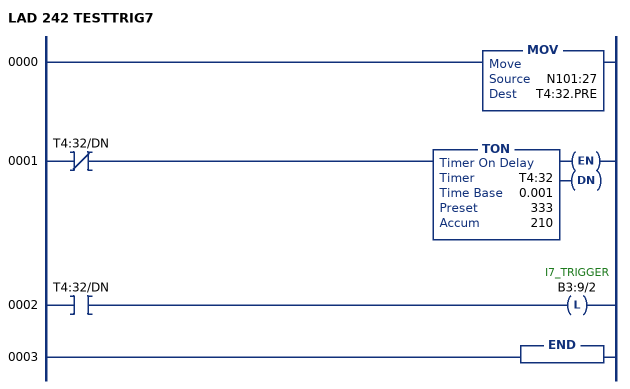
% Rung: 0 %
SOR MOV N101:27 T4:32.PRE EOR
%   N101:27  I7_TRIGTIME %
% Rung: 1 %
SOR XIO T4:32/DN TON T4:32 0.001 333 210 EOR
% Rung: 2 %
SOR XIC T4:32/DN OTL B3:9/2 EOR
%   B3:9/2  I7_TRIGGER %
% Rung: 3 %
SOR END EOR

LADDER 243 "TESTTRIG8"
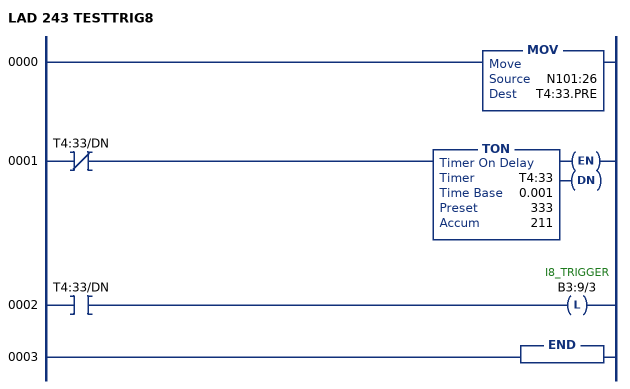
% Rung: 0 %
SOR MOV N101:26 T4:33.PRE EOR
%   N101:26  I8_TRIGTIME %
% Rung: 1 %
SOR XIO T4:33/DN TON T4:33 0.001 333 211 EOR
% Rung: 2 %
SOR XIC T4:33/DN OTL B3:9/3 EOR
%   B3:9/3  I8_TRIGGER %
% Rung: 3 %
SOR END EOR

LADDER 244 "PACKAGER"    % normal %
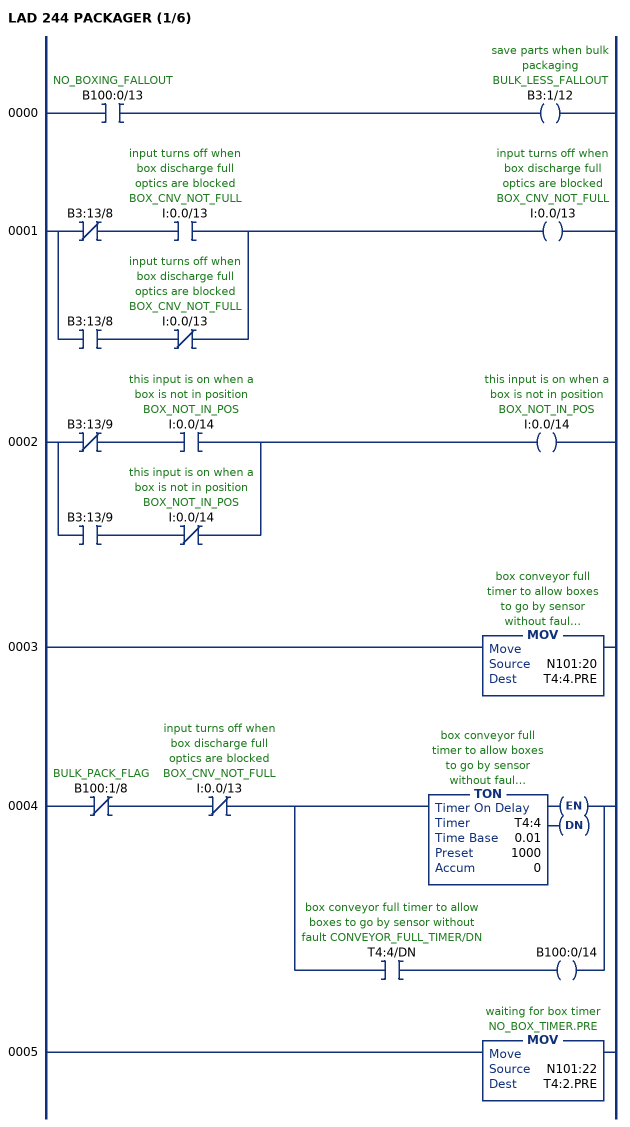
% Rung: 0 %
SOR XIC B100:0/13 OTE B3:1/12 EOR
%   B100:0/13  NO_BOXING_FALLOUT %
%   B3:1/12  BULK_LESS_FALLOUT  "save parts when bulk packaging" %
% Rung: 1 %
SOR BST XIO B3:13/8 XIC I:0.0/13 NXB XIC B3:13/8 XIO I:0.0/13 BND OTE I:0.0/13 EOR
%   I:0.0/13  BOX_CNV_NOT_FULL  "input turns off when box discharge full optics are blocked" %
% Rung: 2 %
SOR BST XIO B3:13/9 XIC I:0.0/14 NXB XIC B3:13/9 XIO I:0.0/14 BND OTE I:0.0/14 EOR
%   I:0.0/14  BOX_NOT_IN_POS  "this input is on when a box is not in position" %
% Rung: 3 %
SOR MOV N101:20 T4:4.PRE EOR
%   N101:20  CONV_FULL_TIME_LIMIT  "time to allow box to pass box conveyor full sensor without fault" %
%   T4:4  CONVEYOR_FULL_TIMER  "box conveyor full timer to allow boxes to go by sensor without fault" %
% Rung: 4 %
SOR XIO B100:1/8 XIO I:0.0/13 BST TON T4:4 0.01 1000 0 NXB XIC T4:4/DN OTE B100:0/14 BND EOR
%   B100:1/8  BULK_PACK_FLAG %
%   I:0.0/13  BOX_CNV_NOT_FULL  "input turns off when box discharge full optics are blocked" %
%   T4:4  CONVEYOR_FULL_TIMER  "box conveyor full timer to allow boxes to go by sensor without fault" %
% Rung: 5 %
SOR MOV N101:22 T4:2.PRE EOR
%   N101:22  BOX_WAIT_TIME_LIMIT  "the time until waiting for box message in hmi (fault)" %
%   T4:2  NO_BOX_TIMER  "waiting for box timer" %

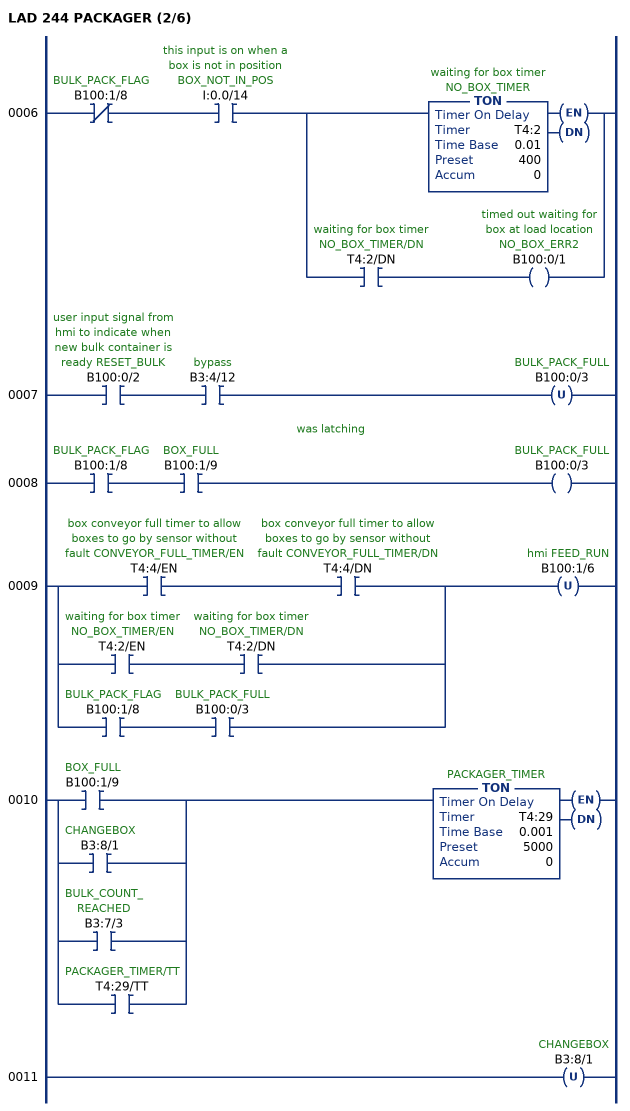
% Rung: 6 %
SOR XIO B100:1/8 XIC I:0.0/14 BST TON T4:2 0.01 400 0 NXB XIC T4:2/DN OTE B100:0/1 BND EOR
%   B100:1/8  BULK_PACK_FLAG %
%   I:0.0/14  BOX_NOT_IN_POS  "this input is on when a box is not in position" %
%   T4:2  NO_BOX_TIMER  "waiting for box timer" %
%   B100:0/1  NO_BOX_ERR2  "timed out waiting for box at load location" %
% Rung: 7 %
SOR XIC B100:0/2 XIC B3:4/12 OTU B100:0/3 EOR
%   B100:0/2  RESET_BULK  "user input signal from hmi to indicate when new bulk container is ready" %
%   B3:4/12  "bypass" %
%   B100:0/3  BULK_PACK_FULL %
% Rung: 8 %
% was latching %
SOR XIC B100:1/8 XIC B100:1/9 OTE B100:0/3 EOR
%   B100:1/8  BULK_PACK_FLAG %
%   B100:1/9  BOX_FULL %
%   B100:0/3  BULK_PACK_FULL %
% Rung: 9 %
SOR BST XIC T4:4/EN XIC T4:4/DN NXB XIC T4:2/EN XIC T4:2/DN NXB XIC B100:1/8 XIC B100:0/3 BND OTU B100:1/6 EOR
%   T4:4  CONVEYOR_FULL_TIMER  "box conveyor full timer to allow boxes to go by sensor without fault" %
%   T4:2  NO_BOX_TIMER  "waiting for box timer" %
%   B100:1/8  BULK_PACK_FLAG %
%   B100:0/3  BULK_PACK_FULL %
%   B100:1/6  FEED_RUN  "hmi" %
% Rung: 10 %
SOR BST XIC B100:1/9 NXB XIC B3:8/1 NXB XIC B3:7/3 NXB XIC T4:29/TT BND TON T4:29 0.001 5000 0 EOR
%   B100:1/9  BOX_FULL %
%   B3:8/1  CHANGEBOX %
%   B3:7/3  BULK_COUNT_REACHED %
%   T4:29  PACKAGER_TIMER %
% Rung: 11 %
SOR OTU B3:8/1 EOR
%   B3:8/1  CHANGEBOX %

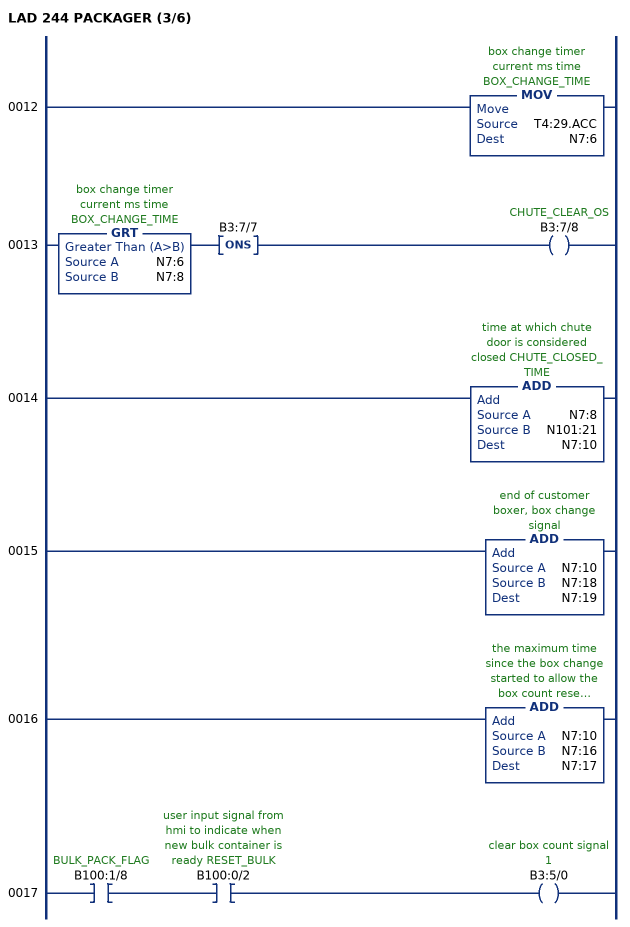
% Rung: 12 %
SOR MOV T4:29.ACC N7:6 EOR
%   T4:29  PACKAGER_TIMER %
%   N7:6  BOX_CHANGE_TIME  "box change timer current ms time" %
% Rung: 13 %
SOR GRT N7:6 N7:8 ONS B3:7/7 OTE B3:7/8 EOR
%   N7:6  BOX_CHANGE_TIME  "box change timer current ms time" %
%   N7:8  CHUTE_CLEAR_TIME %
%   B3:7/8  CHUTE_CLEAR_OS %
% Rung: 14 %
SOR ADD N7:8 N101:21 N7:10 EOR
%   N7:8  CHUTE_CLEAR_TIME %
%   N101:21  CHUTE_CLOSE_TIME  "ms time required to close chute" %
%   N7:10  CHUTE_CLOSED_TIME  "time at which chute door is considered closed" %
% Rung: 15 %
SOR ADD N7:10 N7:18 N7:19 EOR
%   N7:10  CHUTE_CLOSED_TIME  "time at which chute door is considered closed" %
%   N7:18  CHANGE_BOX_SIG_TIME  "customer boxer change box signal time" %
%   N7:19  "end of customer boxer, box change signal" %
% Rung: 16 %
SOR ADD N7:10 N7:16 N7:17 EOR
%   N7:10  CHUTE_CLOSED_TIME  "time at which chute door is considered closed" %
%   N7:16  RESET_COUNT_SIG_TIME  "maximum length of time to hold box count reset signal on" %
%   N7:17  "the maximum time since the box change started to allow the box count reset signal" %
% Rung: 17 %
SOR XIC B100:1/8 XIC B100:0/2 OTE B3:5/0 EOR
%   B100:1/8  BULK_PACK_FLAG %
%   B100:0/2  RESET_BULK  "user input signal from hmi to indicate when new bulk container is ready" %
%   B3:5/0  "clear box count signal 1" %

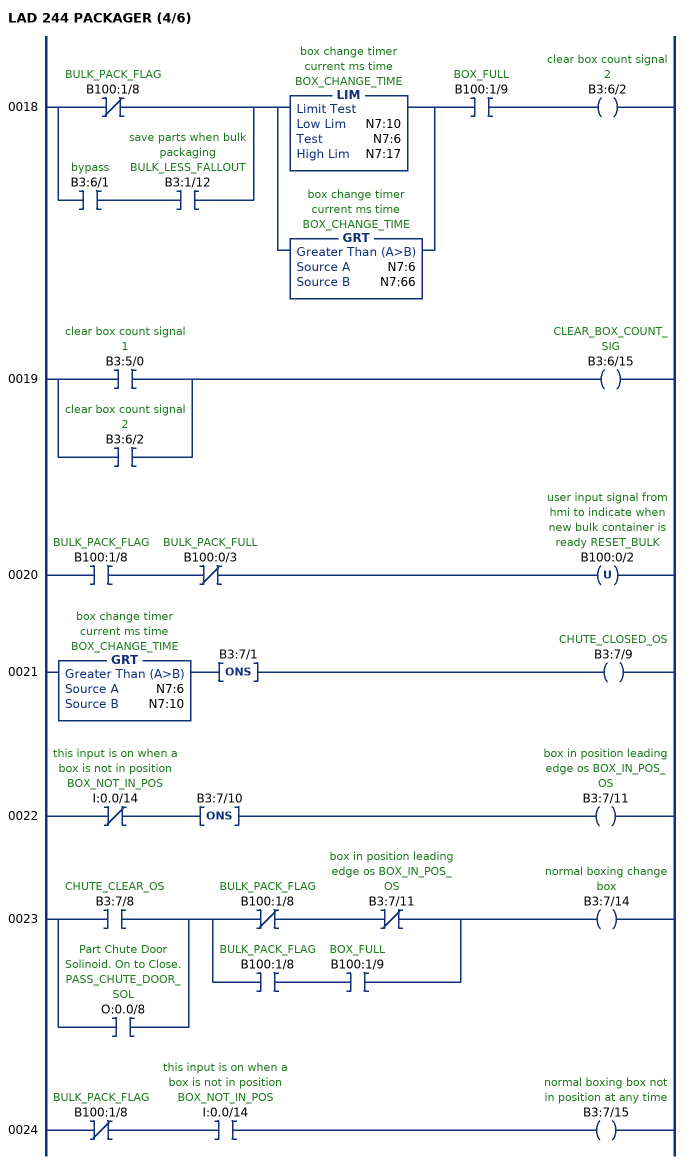
% Rung: 18 %
SOR BST XIO B100:1/8 NXB XIC B3:6/1 XIC B3:1/12 BND BST LIM N7:10 N7:6 N7:17 NXB GRT N7:6 N7:66 BND XIC B100:1/9 OTE B3:6/2 EOR
%   B100:1/8  BULK_PACK_FLAG %
%   B3:6/1  "bypass" %
%   B3:1/12  BULK_LESS_FALLOUT  "save parts when bulk packaging" %
%   N7:10  CHUTE_CLOSED_TIME  "time at which chute door is considered closed" %
%   N7:6  BOX_CHANGE_TIME  "box change timer current ms time" %
%   N7:17  "the maximum time since the box change started to allow the box count reset signal" %
%   B100:1/9  BOX_FULL %
%   B3:6/2  "clear box count signal 2" %
% Rung: 19 %
SOR BST XIC B3:5/0 NXB XIC B3:6/2 BND OTE B3:6/15 EOR
%   B3:5/0  "clear box count signal 1" %
%   B3:6/2  "clear box count signal 2" %
%   B3:6/15  CLEAR_BOX_COUNT_SIG %
% Rung: 20 %
SOR XIC B100:1/8 XIO B100:0/3 OTU B100:0/2 EOR
%   B100:1/8  BULK_PACK_FLAG %
%   B100:0/3  BULK_PACK_FULL %
%   B100:0/2  RESET_BULK  "user input signal from hmi to indicate when new bulk container is ready" %
% Rung: 21 %
SOR GRT N7:6 N7:10 ONS B3:7/1 OTE B3:7/9 EOR
%   N7:6  BOX_CHANGE_TIME  "box change timer current ms time" %
%   N7:10  CHUTE_CLOSED_TIME  "time at which chute door is considered closed" %
%   B3:7/9  CHUTE_CLOSED_OS %
% Rung: 22 %
SOR XIO I:0.0/14 ONS B3:7/10 OTE B3:7/11 EOR
%   I:0.0/14  BOX_NOT_IN_POS  "this input is on when a box is not in position" %
%   B3:7/11  BOX_IN_POS_OS  "box in position leading edge os" %
% Rung: 23 %
SOR BST XIC B3:7/8 NXB XIC O:0.0/8 BND BST XIO B100:1/8 XIO B3:7/11 NXB XIC B100:1/8 XIC B100:1/9 BND OTE B3:7/14 EOR
%   B3:7/8  CHUTE_CLEAR_OS %
%   O:0.0/8  PASS_CHUTE_DOOR_SOL  "Part Chute Door Solinoid. On to Close." %
%   B100:1/8  BULK_PACK_FLAG %
%   B3:7/11  BOX_IN_POS_OS  "box in position leading edge os" %
%   B100:1/9  BOX_FULL %
%   B3:7/14  "normal boxing change box" %
% Rung: 24 %
SOR XIO B100:1/8 XIC I:0.0/14 OTE B3:7/15 EOR
%   B100:1/8  BULK_PACK_FLAG %
%   I:0.0/14  BOX_NOT_IN_POS  "this input is on when a box is not in position" %
%   B3:7/15  "normal boxing box not in position at any time" %

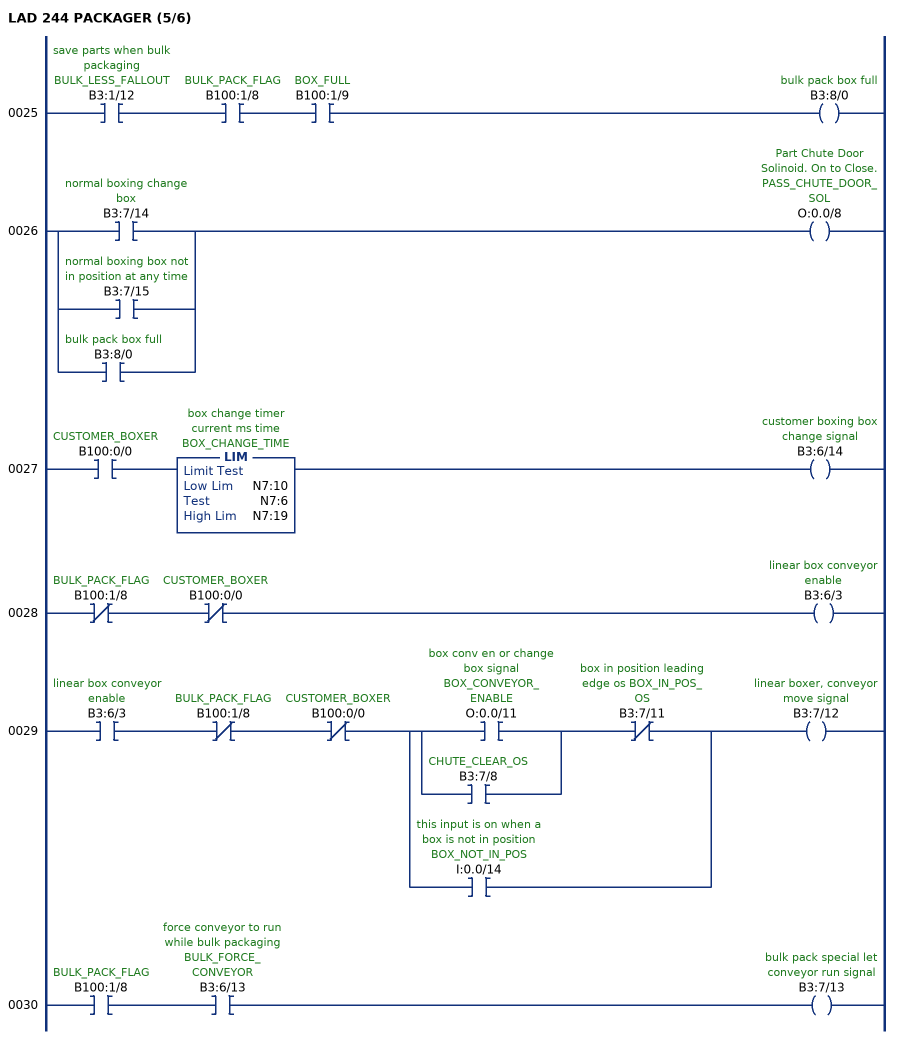
% Rung: 25 %
SOR XIC B3:1/12 XIC B100:1/8 XIC B100:1/9 OTE B3:8/0 EOR
%   B3:1/12  BULK_LESS_FALLOUT  "save parts when bulk packaging" %
%   B100:1/8  BULK_PACK_FLAG %
%   B100:1/9  BOX_FULL %
%   B3:8/0  "bulk pack box full" %
% Rung: 26 %
SOR BST XIC B3:7/14 NXB XIC B3:7/15 NXB XIC B3:8/0 BND OTE O:0.0/8 EOR
%   B3:7/14  "normal boxing change box" %
%   B3:7/15  "normal boxing box not in position at any time" %
%   B3:8/0  "bulk pack box full" %
%   O:0.0/8  PASS_CHUTE_DOOR_SOL  "Part Chute Door Solinoid. On to Close." %
% Rung: 27 %
SOR XIC B100:0/0 LIM N7:10 N7:6 N7:19 OTE B3:6/14 EOR
%   B100:0/0  CUSTOMER_BOXER %
%   N7:10  CHUTE_CLOSED_TIME  "time at which chute door is considered closed" %
%   N7:6  BOX_CHANGE_TIME  "box change timer current ms time" %
%   N7:19  "end of customer boxer, box change signal" %
%   B3:6/14  "customer boxing box change signal" %
% Rung: 28 %
SOR XIO B100:1/8 XIO B100:0/0 OTE B3:6/3 EOR
%   B100:1/8  BULK_PACK_FLAG %
%   B100:0/0  CUSTOMER_BOXER %
%   B3:6/3  "linear box conveyor enable" %
% Rung: 29 %
SOR XIC B3:6/3 XIO B100:1/8 XIO B100:0/0 BST BST XIC O:0.0/11 NXB XIC B3:7/8 BND XIO B3:7/11 NXB XIC I:0.0/14 BND OTE B3:7/12 EOR
%   B3:6/3  "linear box conveyor enable" %
%   B100:1/8  BULK_PACK_FLAG %
%   B100:0/0  CUSTOMER_BOXER %
%   O:0.0/11  BOX_CONVEYOR_ENABLE  "box conv en or change box signal" %
%   B3:7/8  CHUTE_CLEAR_OS %
%   B3:7/11  BOX_IN_POS_OS  "box in position leading edge os" %
%   I:0.0/14  BOX_NOT_IN_POS  "this input is on when a box is not in position" %
%   B3:7/12  "linear boxer, conveyor move signal" %
% Rung: 30 %
SOR XIC B100:1/8 XIC B3:6/13 OTE B3:7/13 EOR
%   B100:1/8  BULK_PACK_FLAG %
%   B3:6/13  BULK_FORCE_CONVEYOR  "force conveyor to run while bulk packaging" %
%   B3:7/13  "bulk pack special let conveyor run signal" %

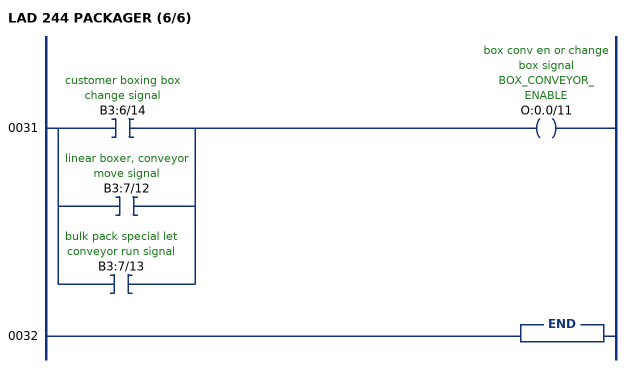
% Rung: 31 %
SOR BST XIC B3:6/14 NXB XIC B3:7/12 NXB XIC B3:7/13 BND OTE O:0.0/11 EOR
%   B3:6/14  "customer boxing box change signal" %
%   B3:7/12  "linear boxer, conveyor move signal" %
%   B3:7/13  "bulk pack special let conveyor run signal" %
%   O:0.0/11  BOX_CONVEYOR_ENABLE  "box conv en or change box signal" %
% Rung: 32 %
SOR END EOR

LADDER 245 "NO PACKAGE"
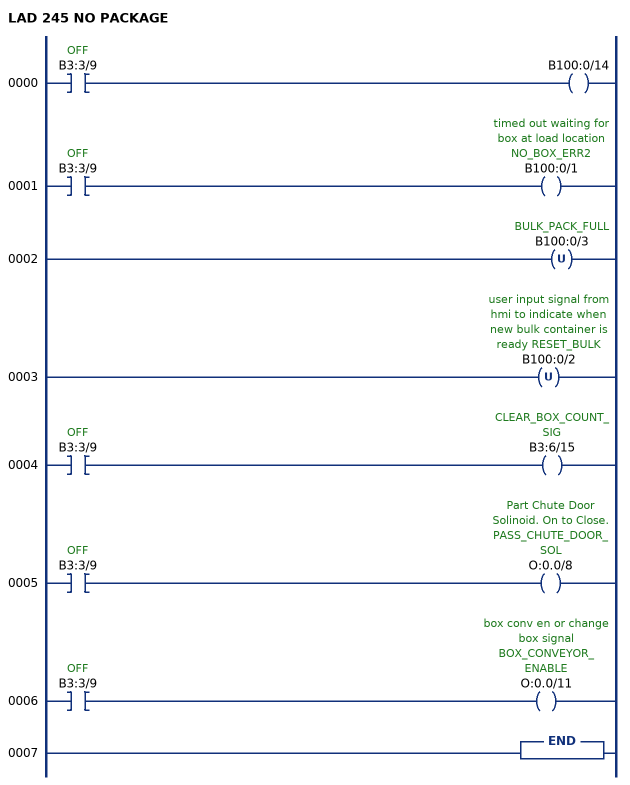
% Rung: 0 %
SOR XIC B3:3/9 OTE B100:0/14 EOR
%   B3:3/9  OFF %
% Rung: 1 %
SOR XIC B3:3/9 OTE B100:0/1 EOR
%   B3:3/9  OFF %
%   B100:0/1  NO_BOX_ERR2  "timed out waiting for box at load location" %
% Rung: 2 %
SOR OTU B100:0/3 EOR
%   B100:0/3  BULK_PACK_FULL %
% Rung: 3 %
SOR OTU B100:0/2 EOR
%   B100:0/2  RESET_BULK  "user input signal from hmi to indicate when new bulk container is ready" %
% Rung: 4 %
SOR XIC B3:3/9 OTE B3:6/15 EOR
%   B3:3/9  OFF %
%   B3:6/15  CLEAR_BOX_COUNT_SIG %
% Rung: 5 %
SOR XIC B3:3/9 OTE O:0.0/8 EOR
%   B3:3/9  OFF %
%   O:0.0/8  PASS_CHUTE_DOOR_SOL  "Part Chute Door Solinoid. On to Close." %
% Rung: 6 %
SOR XIC B3:3/9 OTE O:0.0/11 EOR
%   B3:3/9  OFF %
%   O:0.0/11  BOX_CONVEYOR_ENABLE  "box conv en or change box signal" %
% Rung: 7 %
SOR END EOR

LADDER 246 "RATE1"
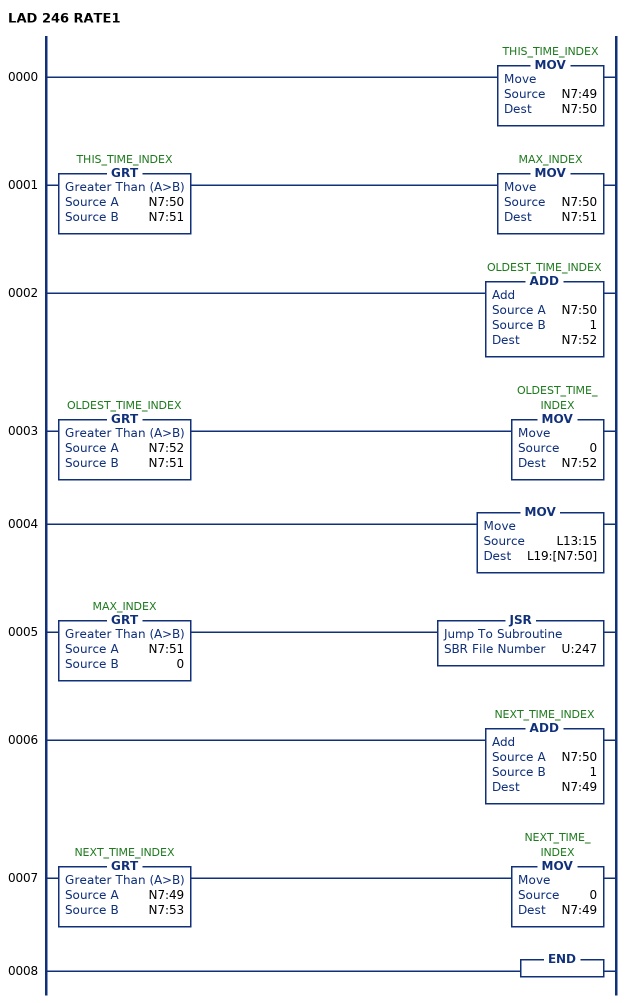
% Rung: 0 %
SOR MOV N7:49 N7:50 EOR
%   N7:49  NEXT_TIME_INDEX %
%   N7:50  THIS_TIME_INDEX %
% Rung: 1 %
SOR GRT N7:50 N7:51 MOV N7:50 N7:51 EOR
%   N7:50  THIS_TIME_INDEX %
%   N7:51  MAX_INDEX %
% Rung: 2 %
SOR ADD N7:50 1 N7:52 EOR
%   N7:50  THIS_TIME_INDEX %
%   N7:52  OLDEST_TIME_INDEX %
% Rung: 3 %
SOR GRT N7:52 N7:51 MOV 0 N7:52 EOR
%   N7:52  OLDEST_TIME_INDEX %
%   N7:51  MAX_INDEX %
% Rung: 4 %
SOR MOV L13:15 L19:[N7:50] EOR
%   L13:15  THE_TIME %
%   N7:50  THIS_TIME_INDEX %
% Rung: 5 %
SOR GRT N7:51 0 JSR U:247 EOR
%   N7:51  MAX_INDEX %
% Rung: 6 %
SOR ADD N7:50 1 N7:49 EOR
%   N7:50  THIS_TIME_INDEX %
%   N7:49  NEXT_TIME_INDEX %
% Rung: 7 %
SOR GRT N7:49 N7:53 MOV 0 N7:49 EOR
%   N7:49  NEXT_TIME_INDEX %
%   N7:53  UPPER_INDEX_LIMIT %
% Rung: 8 %
SOR END EOR

LADDER 247 "RATE2"
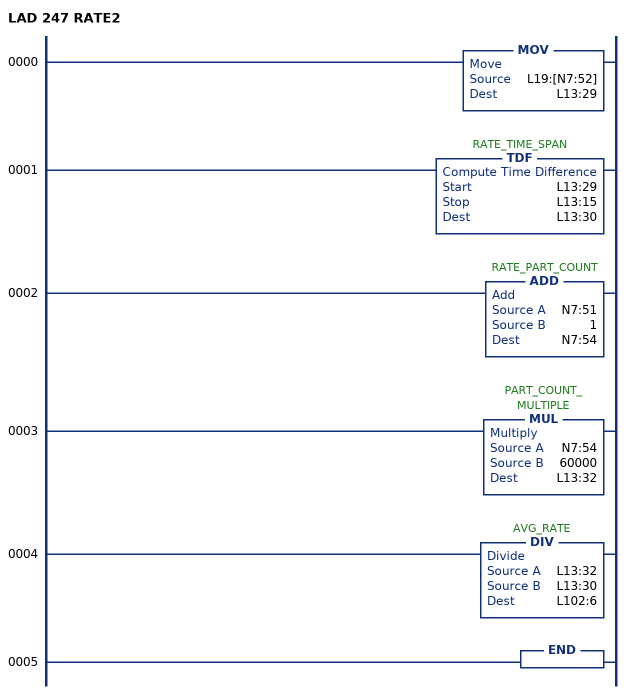
% Rung: 0 %
SOR MOV L19:[N7:52] L13:29 EOR
%   N7:52  OLDEST_TIME_INDEX %
% Rung: 1 %
SOR TDF L13:29 L13:15 L13:30 EOR
%   L13:15  THE_TIME %
%   L13:30  RATE_TIME_SPAN %
% Rung: 2 %
SOR ADD N7:51 1 N7:54 EOR
%   N7:51  MAX_INDEX %
%   N7:54  RATE_PART_COUNT %
% Rung: 3 %
SOR MUL N7:54 60000 L13:32 EOR
%   N7:54  RATE_PART_COUNT %
%   L13:32  PART_COUNT_MULTIPLE %
% Rung: 4 %
SOR DIV L13:32 L13:30 L102:6 EOR
%   L13:32  PART_COUNT_MULTIPLE %
%   L13:30  RATE_TIME_SPAN %
%   L102:6  AVG_RATE %
% Rung: 5 %
SOR END EOR

LADDER 248 "RESET RATE"
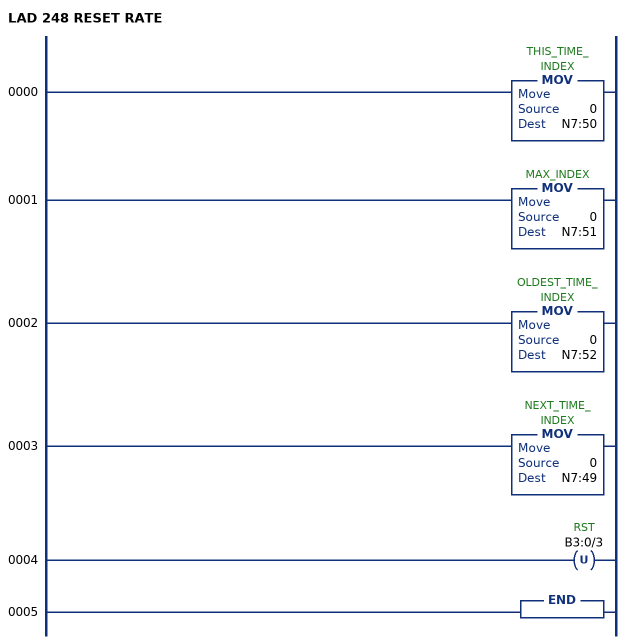
% Rung: 0 %
SOR MOV 0 N7:50 EOR
%   N7:50  THIS_TIME_INDEX %
% Rung: 1 %
SOR MOV 0 N7:51 EOR
%   N7:51  MAX_INDEX %
% Rung: 2 %
SOR MOV 0 N7:52 EOR
%   N7:52  OLDEST_TIME_INDEX %
% Rung: 3 %
SOR MOV 0 N7:49 EOR
%   N7:49  NEXT_TIME_INDEX %
% Rung: 4 %
SOR OTU B3:0/3 EOR
%   B3:0/3  RST %
% Rung: 5 %
SOR END EOR

LADDER 249 "NP STOP"    % stop on no good %
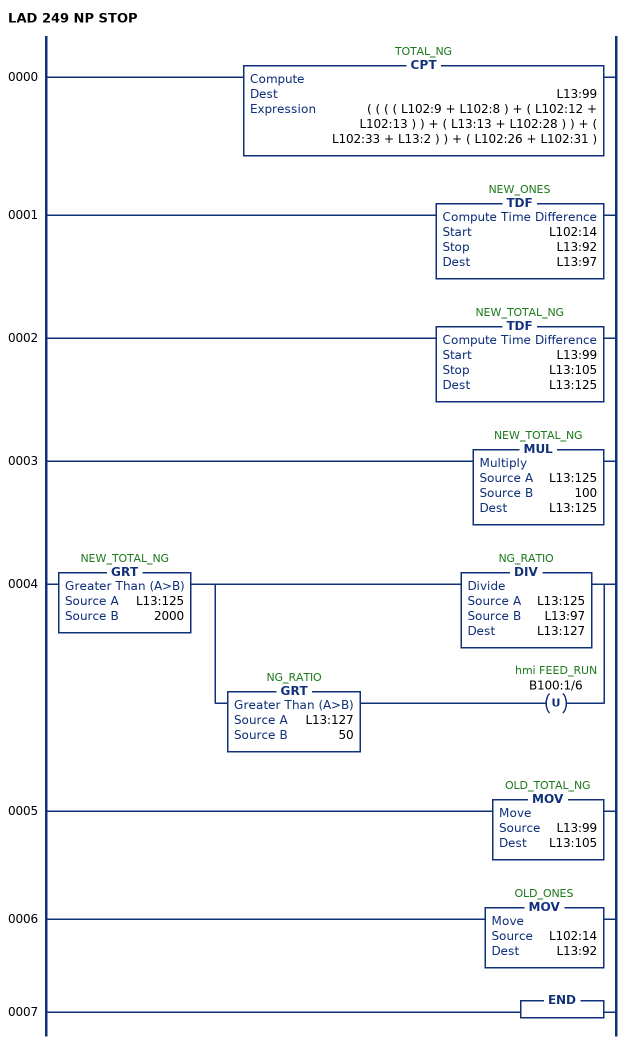
% Rung: 0 %
SOR CPT L13:99 " ( ( ( ( L102:9 + L102:8 ) + ( L102:12 + L102:13 ) ) + ( L13:13 + L102:28 ) ) + ( L102:33 + L13:2 ) ) + ( L102:26 + L102:31 ) " EOR
%   L13:99  TOTAL_NG %
%   L102:9  "too wide bottom" %
%   L102:8  "too close bottom" %
%   L102:12  "too close top count" %
%   L102:13  "too wide top count" %
%   L102:28  I1_I5_SKIPPEDCOUNT %
%   L102:33  I2_I6_SKIPPEDCOUNT %
%   L102:26  I1_I5_FAIL_COUNT %
%   L102:31  I2_I6_FAIL_COUNT %
% Rung: 1 %
SOR TDF L102:14 L13:92 L13:97 EOR
%   L102:14  ONES %
%   L13:92  OLD_ONES %
%   L13:97  NEW_ONES %
% Rung: 2 %
SOR TDF L13:99 L13:105 L13:125 EOR
%   L13:99  TOTAL_NG %
%   L13:105  OLD_TOTAL_NG %
%   L13:125  NEW_TOTAL_NG %
% Rung: 3 %
SOR MUL L13:125 100 L13:125 EOR
%   L13:125  NEW_TOTAL_NG %
% Rung: 4 %
SOR GRT L13:125 2000 BST DIV L13:125 L13:97 L13:127 NXB GRT L13:127 50 OTU B100:1/6 BND EOR
%   L13:125  NEW_TOTAL_NG %
%   L13:97  NEW_ONES %
%   L13:127  NG_RATIO %
%   B100:1/6  FEED_RUN  "hmi" %
% Rung: 5 %
SOR MOV L13:99 L13:105 EOR
%   L13:99  TOTAL_NG %
%   L13:105  OLD_TOTAL_NG %
% Rung: 6 %
SOR MOV L102:14 L13:92 EOR
%   L102:14  ONES %
%   L13:92  OLD_ONES %
% Rung: 7 %
SOR END EOR

LADDER 250 "SPEED BOT"    % high speed %
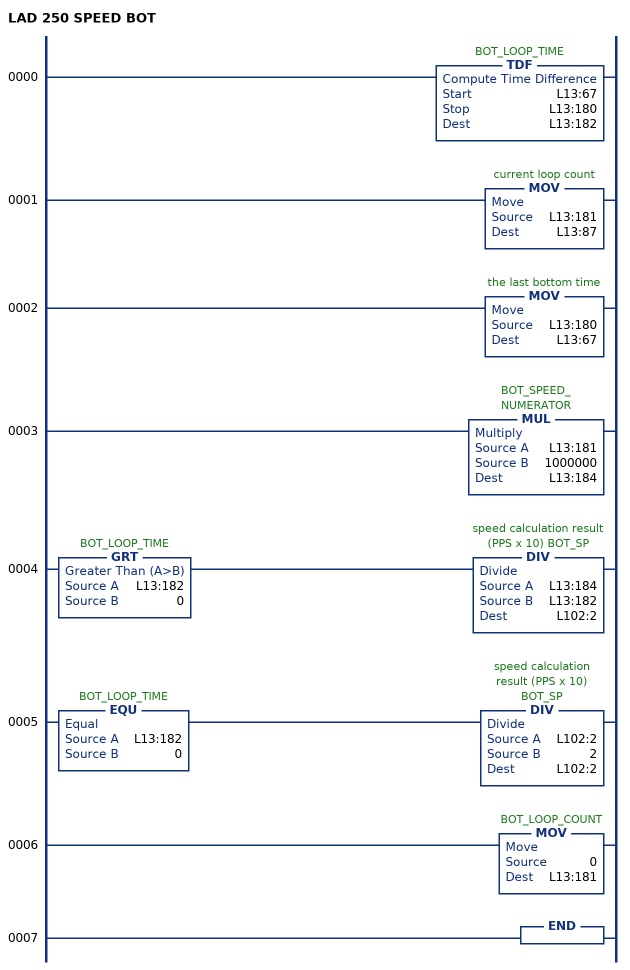
% Rung: 0 %
SOR TDF L13:67 L13:180 L13:182 EOR
%   L13:67  "the last bottom time" %
%   L13:180  BOT_THIS_TIME  "rtc bot belt movement event time" %
%   L13:182  BOT_LOOP_TIME %
% Rung: 1 %
SOR MOV L13:181 L13:87 EOR
%   L13:181  BOT_LOOP_COUNT %
%   L13:87  "current loop count" %
% Rung: 2 %
SOR MOV L13:180 L13:67 EOR
%   L13:180  BOT_THIS_TIME  "rtc bot belt movement event time" %
%   L13:67  "the last bottom time" %
% Rung: 3 %
SOR MUL L13:181 1000000 L13:184 EOR
%   L13:181  BOT_LOOP_COUNT %
%   L13:184  BOT_SPEED_NUMERATOR %
% Rung: 4 %
SOR GRT L13:182 0 DIV L13:184 L13:182 L102:2 EOR
%   L13:182  BOT_LOOP_TIME %
%   L13:184  BOT_SPEED_NUMERATOR %
%   L102:2  BOT_SP  "speed calculation result (PPS x 10)" %
% Rung: 5 %
SOR EQU L13:182 0 DIV L102:2 2 L102:2 EOR
%   L13:182  BOT_LOOP_TIME %
%   L102:2  BOT_SP  "speed calculation result (PPS x 10)" %
% Rung: 6 %
SOR MOV 0 L13:181 EOR
%   L13:181  BOT_LOOP_COUNT %
% Rung: 7 %
SOR END EOR

LADDER 251 "SPEED TOP"    % high speed %
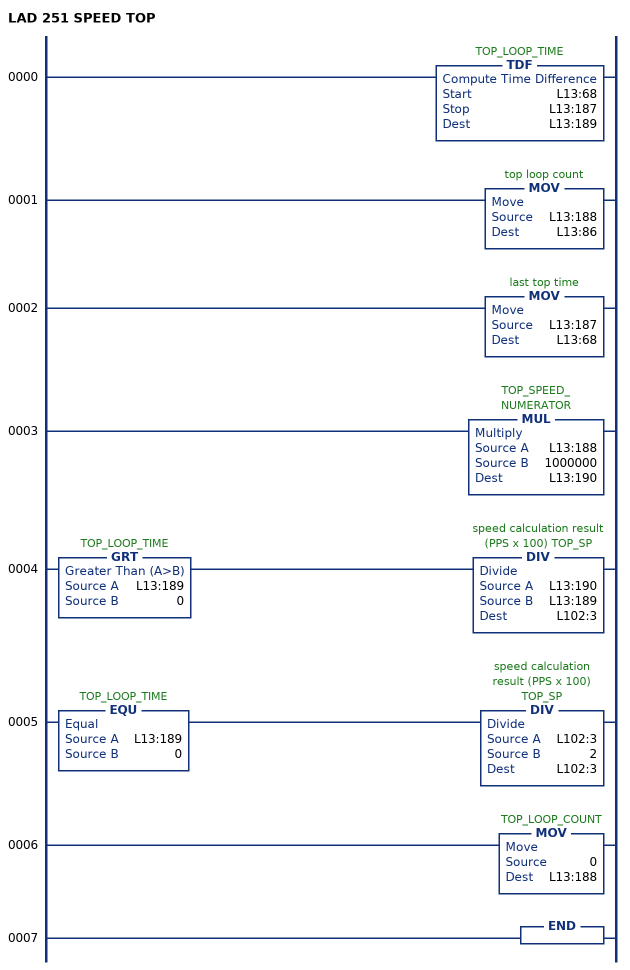
% Rung: 0 %
SOR TDF L13:68 L13:187 L13:189 EOR
%   L13:68  "last top time" %
%   L13:187  TOP_THIS_TIME  "rtc top belt movement event time" %
%   L13:189  TOP_LOOP_TIME %
% Rung: 1 %
SOR MOV L13:188 L13:86 EOR
%   L13:188  TOP_LOOP_COUNT %
%   L13:86  "top loop count" %
% Rung: 2 %
SOR MOV L13:187 L13:68 EOR
%   L13:187  TOP_THIS_TIME  "rtc top belt movement event time" %
%   L13:68  "last top time" %
% Rung: 3 %
SOR MUL L13:188 1000000 L13:190 EOR
%   L13:188  TOP_LOOP_COUNT %
%   L13:190  TOP_SPEED_NUMERATOR %
% Rung: 4 %
SOR GRT L13:189 0 DIV L13:190 L13:189 L102:3 EOR
%   L13:189  TOP_LOOP_TIME %
%   L13:190  TOP_SPEED_NUMERATOR %
%   L102:3  TOP_SP  "speed calculation result (PPS x 100)" %
% Rung: 5 %
SOR EQU L13:189 0 DIV L102:3 2 L102:3 EOR
%   L13:189  TOP_LOOP_TIME %
%   L102:3  TOP_SP  "speed calculation result (PPS x 100)" %
% Rung: 6 %
SOR MOV 0 L13:188 EOR
%   L13:188  TOP_LOOP_COUNT %
% Rung: 7 %
SOR END EOR

LADDER 252 "P BOT"    % high speed %
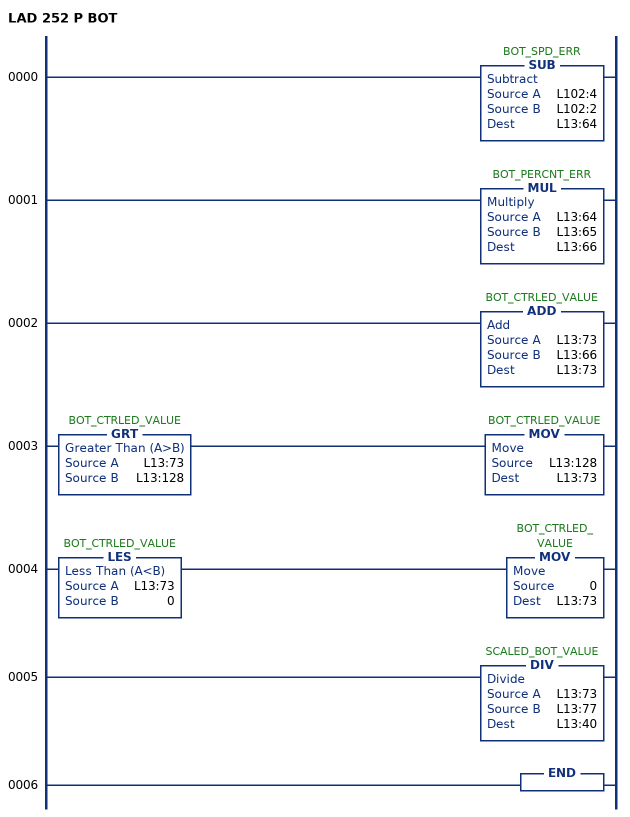
% Rung: 0 %
SOR SUB L102:4 L102:2 L13:64 EOR
%   L102:4  BOT_SPD_SETPOINT %
%   L102:2  BOT_SP  "speed calculation result (PPS x 10)" %
%   L13:64  BOT_SPD_ERR %
% Rung: 1 %
SOR MUL L13:64 L13:65 L13:66 EOR
%   L13:64  BOT_SPD_ERR %
%   L13:65  POS5SHIFT %
%   L13:66  BOT_PERCNT_ERR %
% Rung: 2 %
SOR ADD L13:73 L13:66 L13:73 EOR
%   L13:73  BOT_CTRLED_VALUE %
%   L13:66  BOT_PERCNT_ERR %
% Rung: 3 %
SOR GRT L13:73 L13:128 MOV L13:128 L13:73 EOR
%   L13:73  BOT_CTRLED_VALUE %
%   L13:128  "how much top has shifted since measurment" %
% Rung: 4 %
SOR LES L13:73 0 MOV 0 L13:73 EOR
%   L13:73  BOT_CTRLED_VALUE %
% Rung: 5 %
SOR DIV L13:73 L13:77 L13:40 EOR
%   L13:73  BOT_CTRLED_VALUE %
%   L13:40  SCALED_BOT_VALUE %
% Rung: 6 %
SOR END EOR

LADDER 253 "P TOP"    % high speed %
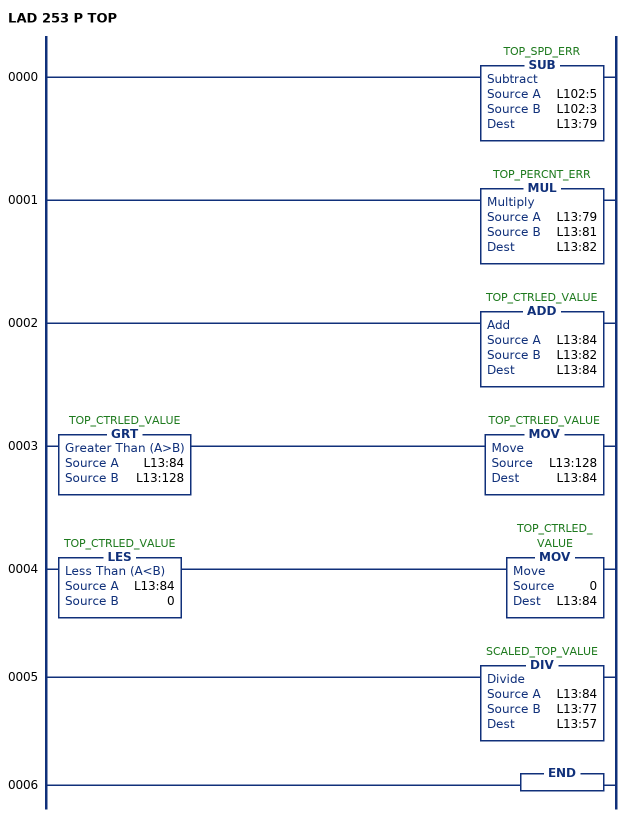
% Rung: 0 %
SOR SUB L102:5 L102:3 L13:79 EOR
%   L102:5  TOP_SPD_SETPOINT %
%   L102:3  TOP_SP  "speed calculation result (PPS x 100)" %
%   L13:79  TOP_SPD_ERR %
% Rung: 1 %
SOR MUL L13:79 L13:81 L13:82 EOR
%   L13:79  TOP_SPD_ERR %
%   L13:81  TOP_FDBK_RATIO %
%   L13:82  TOP_PERCNT_ERR %
% Rung: 2 %
SOR ADD L13:84 L13:82 L13:84 EOR
%   L13:84  TOP_CTRLED_VALUE %
%   L13:82  TOP_PERCNT_ERR %
% Rung: 3 %
SOR GRT L13:84 L13:128 MOV L13:128 L13:84 EOR
%   L13:84  TOP_CTRLED_VALUE %
%   L13:128  "how much top has shifted since measurment" %
% Rung: 4 %
SOR LES L13:84 0 MOV 0 L13:84 EOR
%   L13:84  TOP_CTRLED_VALUE %
% Rung: 5 %
SOR DIV L13:84 L13:77 L13:57 EOR
%   L13:84  TOP_CTRLED_VALUE %
%   L13:57  SCALED_TOP_VALUE %
% Rung: 6 %
SOR END EOR

LADDER 254 "TOTALCOUNT"
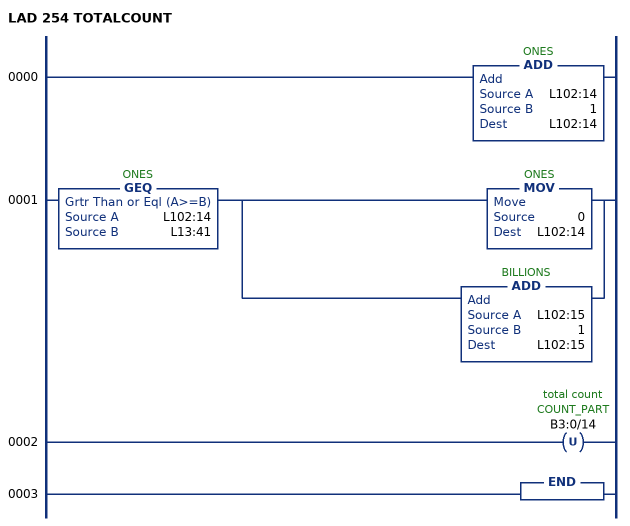
% Rung: 0 %
SOR ADD L102:14 1 L102:14 EOR
%   L102:14  ONES %
% Rung: 1 %
SOR GEQ L102:14 L13:41 BST MOV 0 L102:14 NXB ADD L102:15 1 L102:15 BND EOR
%   L102:14  ONES %
%   L13:41  "skipped count change in the last 3 seconds" %
%   L102:15  BILLIONS %
% Rung: 2 %
SOR OTU B3:0/14 EOR
%   B3:0/14  COUNT_PART  "total count" %
% Rung: 3 %
SOR END EOR

LADDER 255 "SAVED"
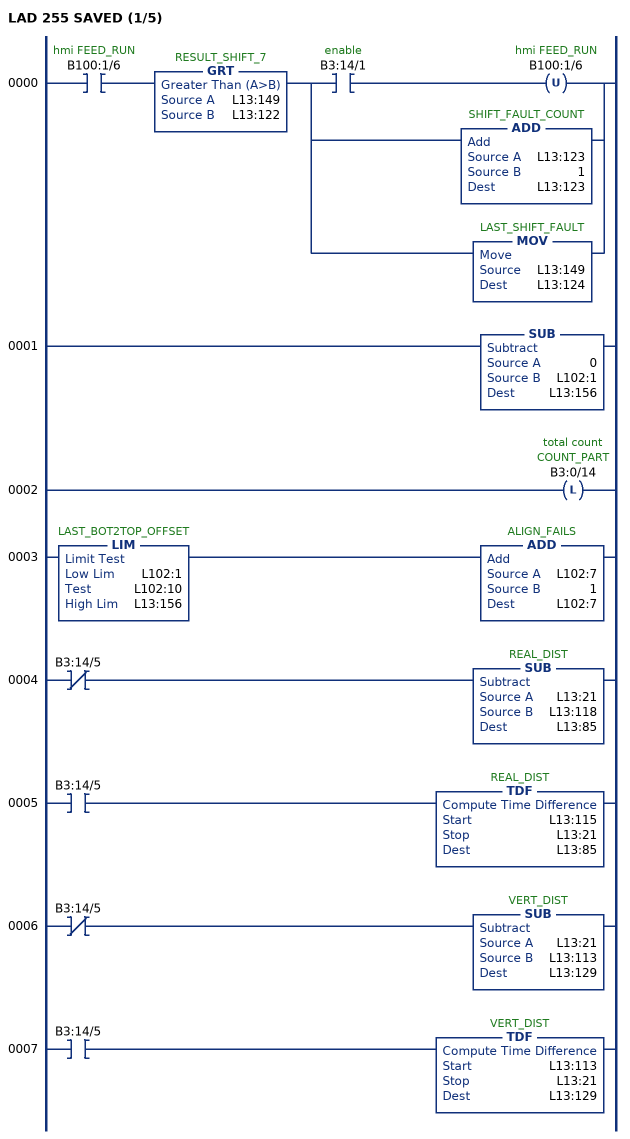
% Rung: 0 %
SOR XIC B100:1/6 GRT L13:149 L13:122 BST XIC B3:14/1 OTU B100:1/6 NXB ADD L13:123 1 L13:123 NXB MOV L13:149 L13:124 BND EOR
%   B100:1/6  FEED_RUN  "hmi" %
%   L13:149  RESULT_SHIFT_7 %
%   L13:122  TOP_SHIFT_FAULT_LIM  "remove me" %
%   B3:14/1  "enable" %
%   L13:123  SHIFT_FAULT_COUNT %
%   L13:124  LAST_SHIFT_FAULT %
% Rung: 1 %
SOR SUB 0 L102:1 L13:156 EOR
%   L102:1  MAX_OFFSET  "transition zone width" %
% Rung: 2 %
SOR OTL B3:0/14 EOR
%   B3:0/14  COUNT_PART  "total count" %
% Rung: 3 %
SOR LIM L102:1 L102:10 L13:156 ADD L102:7 1 L102:7 EOR
%   L102:1  MAX_OFFSET  "transition zone width" %
%   L102:10  LAST_BOT2TOP_OFFSET %
%   L102:7  ALIGN_FAILS %
% Rung: 4 %
SOR XIO B3:14/5 SUB L13:21 L13:118 L13:85 EOR
%   L13:21  TOP_POSITION %
%   L13:118  REAL_CL_POSITION  "real part center line in raw position" %
%   L13:85  REAL_DIST %
% Rung: 5 %
SOR XIC B3:14/5 TDF L13:115 L13:21 L13:85 EOR
%   L13:115  TRAILING_EDGE_POS  "top optic trailing edge position" %
%   L13:21  TOP_POSITION %
%   L13:85  REAL_DIST %
% Rung: 6 %
SOR XIO B3:14/5 SUB L13:21 L13:113 L13:129 EOR
%   L13:21  TOP_POSITION %
%   L13:113  VIRT_CL_POSITION  "virtual part center line transfer from the bottom in raw position" %
%   L13:129  VERT_DIST %
% Rung: 7 %
SOR XIC B3:14/5 TDF L13:113 L13:21 L13:129 EOR
%   L13:113  VIRT_CL_POSITION  "virtual part center line transfer from the bottom in raw position" %
%   L13:21  TOP_POSITION %
%   L13:129  VERT_DIST %

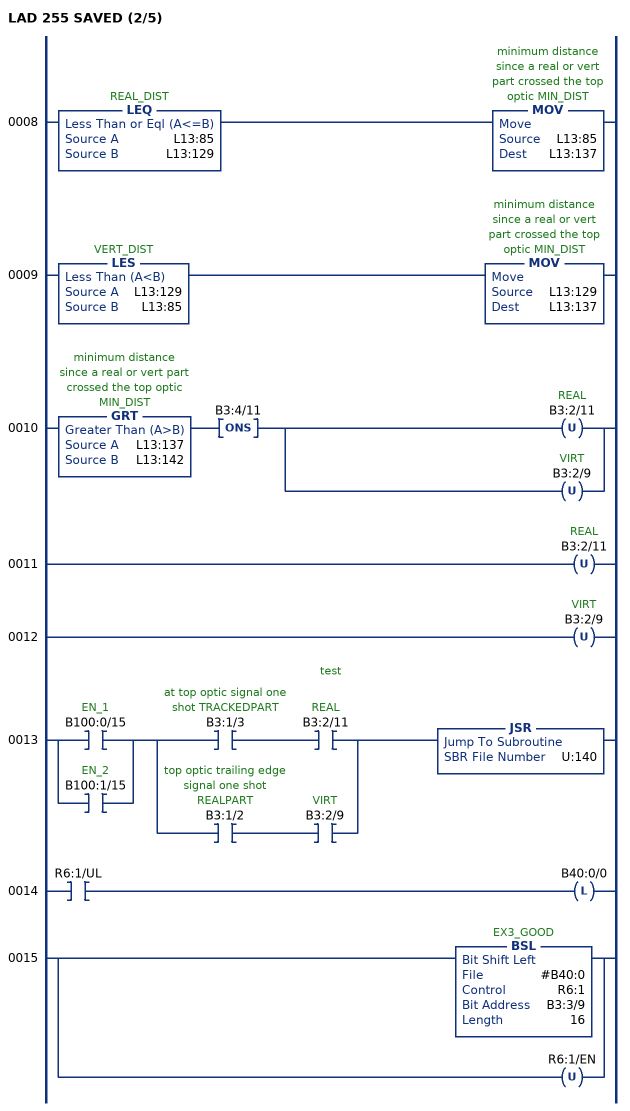
% Rung: 8 %
SOR LEQ L13:85 L13:129 MOV L13:85 L13:137 EOR
%   L13:85  REAL_DIST %
%   L13:129  VERT_DIST %
%   L13:137  MIN_DIST  "minimum distance since a real or vert part crossed the top optic" %
% Rung: 9 %
SOR LES L13:129 L13:85 MOV L13:129 L13:137 EOR
%   L13:129  VERT_DIST %
%   L13:85  REAL_DIST %
%   L13:137  MIN_DIST  "minimum distance since a real or vert part crossed the top optic" %
% Rung: 10 %
SOR GRT L13:137 L13:142 ONS B3:4/11 BST OTU B3:2/11 NXB OTU B3:2/9 BND EOR
%   L13:137  MIN_DIST  "minimum distance since a real or vert part crossed the top optic" %
%   L13:142  LAST_ALIGNMENT_FAILS %
%   B3:2/11  REAL %
%   B3:2/9  VIRT %
% Rung: 11 %
SOR OTU B3:2/11 EOR
%   B3:2/11  REAL %
% Rung: 12 %
SOR OTU B3:2/9 EOR
%   B3:2/9  VIRT %
% Rung: 13 %
% test %
SOR BST XIC B100:0/15 NXB XIC B100:1/15 BND BST XIC B3:1/3 XIC B3:2/11 NXB XIC B3:1/2 XIC B3:2/9 BND JSR U:140 EOR
%   B100:0/15  EN_1 %
%   B100:1/15  EN_2 %
%   B3:1/3  TRACKEDPART  "at top optic signal one shot" %
%   B3:2/11  REAL %
%   B3:1/2  REALPART  "top optic trailing edge signal one shot" %
%   B3:2/9  VIRT %
% Rung: 14 %
SOR XIC R6:1/UL OTL B40:0/0 EOR
% Rung: 15 %
SOR BST BSL #B40:0 R6:1 B3:3/9 16 NXB OTU R6:1/EN BND EOR
%   B40:0  EX3_GOOD %
%   B3:3/9  OFF %

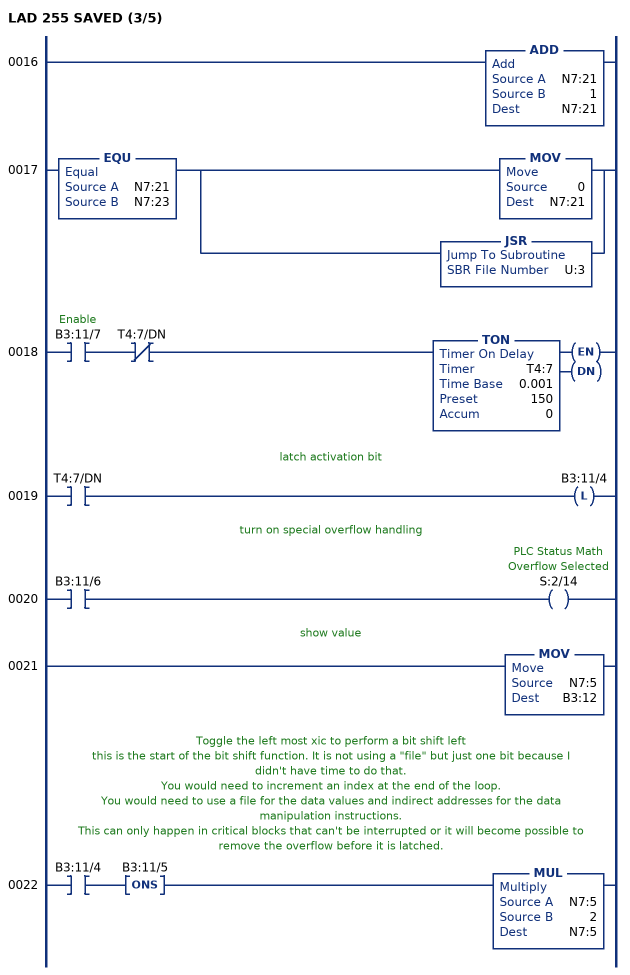
% Rung: 16 %
SOR ADD N7:21 1 N7:21 EOR
% Rung: 17 %
SOR EQU N7:21 N7:23 BST MOV 0 N7:21 NXB JSR U:3 BND EOR
% Rung: 18 %
SOR XIC B3:11/7 XIO T4:7/DN TON T4:7 0.001 150 0 EOR
%   B3:11/7  "Enable" %
% Rung: 19 %
% latch activation bit %
SOR XIC T4:7/DN OTL B3:11/4 EOR
% Rung: 20 %
% turn on special overflow handling %
SOR XIC B3:11/6 OTE S:2/14 EOR
%   S:2/14  "PLC Status Math Overflow Selected" %
% Rung: 21 %
% show value %
SOR MOV N7:5 B3:12 EOR
% Rung: 22 %
% Toggle the left most xic to perform a bit shift left
% 
% this is the start of the bit shift function. It is not using a "file" but just one bit because I didn't have time to do that.
% You would need to increment an index at the end of the loop.
% You would need to use a file for the data values and indirect addresses for the data manipulation instructions.
% 
% This can only happen in critical blocks that can't be interrupted or it will become possible to remove the overflow before it is latched. %
SOR XIC B3:11/4 ONS B3:11/5 MUL N7:5 2 N7:5 EOR

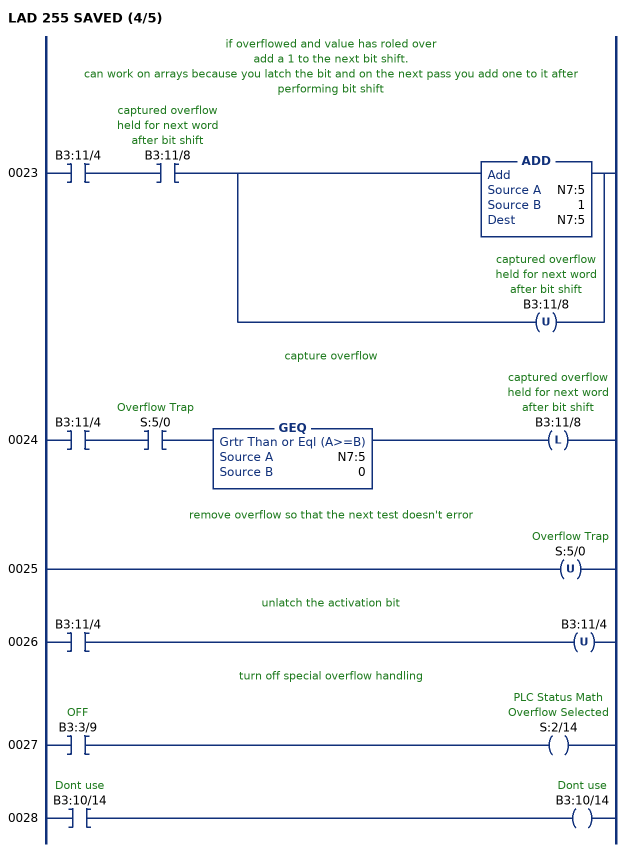
% Rung: 23 %
% if overflowed and value has roled over
% add a 1 to the next bit shift.
% can work on arrays because you latch the bit and on the next pass you add one to it after performing bit shift %
SOR XIC B3:11/4 XIC B3:11/8 BST ADD N7:5 1 N7:5 NXB OTU B3:11/8 BND EOR
%   B3:11/8  "captured overflow held for next word after bit shift" %
% Rung: 24 %
% capture overflow %
SOR XIC B3:11/4 XIC S:5/0 GEQ N7:5 0 OTL B3:11/8 EOR
%   S:5/0  "Overflow Trap" %
%   B3:11/8  "captured overflow held for next word after bit shift" %
% Rung: 25 %
% remove overflow so that the next test doesn't error %
SOR OTU S:5/0 EOR
%   S:5/0  "Overflow Trap" %
% Rung: 26 %
% unlatch the activation bit %
SOR XIC B3:11/4 OTU B3:11/4 EOR
% Rung: 27 %
% turn off special overflow handling %
SOR XIC B3:3/9 OTE S:2/14 EOR
%   B3:3/9  OFF %
%   S:2/14  "PLC Status Math Overflow Selected" %
% Rung: 28 %
SOR XIC B3:10/14 OTE B3:10/14 EOR
%   B3:10/14  "Dont use" %

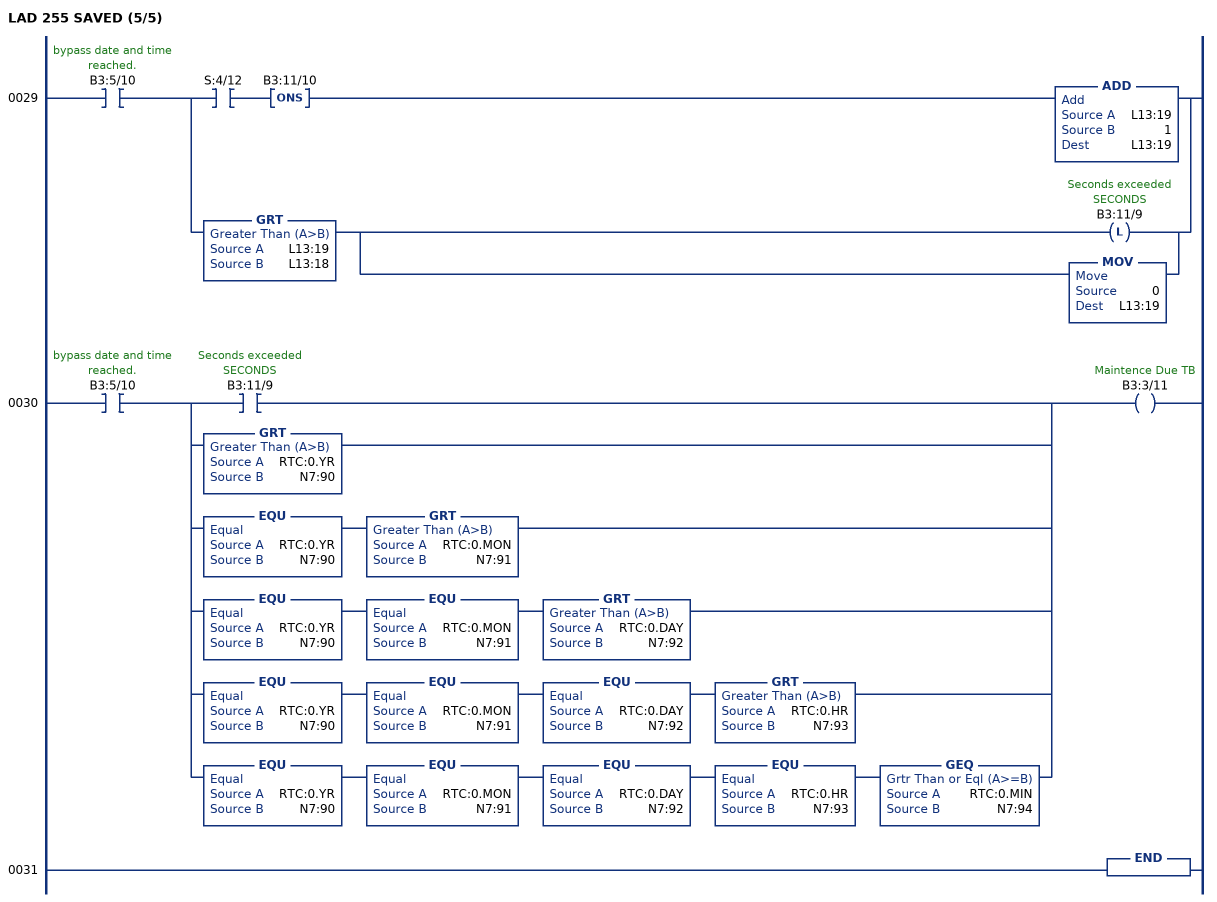
% Rung: 29 %
SOR XIC B3:5/10 BST XIC S:4/12 ONS B3:11/10 ADD L13:19 1 L13:19 NXB GRT L13:19 L13:18 BST OTL B3:11/9 NXB MOV 0 L13:19 BND BND EOR
%   B3:5/10  "bypass date and time reached." %
%   L13:18  MAX %
%   B3:11/9  SECONDS  "Seconds exceeded" %
% Rung: 30 %
SOR XIC B3:5/10 BST XIC B3:11/9 NXB GRT RTC:0.YR N7:90 NXB EQU RTC:0.YR N7:90 GRT RTC:0.MON N7:91 NXB EQU RTC:0.YR N7:90 EQU RTC:0.MON N7:91 GRT RTC:0.DAY N7:92 NXB EQU RTC:0.YR N7:90 EQU RTC:0.MON N7:91 EQU RTC:0.DAY N7:92 GRT RTC:0.HR N7:93 NXB EQU RTC:0.YR N7:90 EQU RTC:0.MON N7:91 EQU RTC:0.DAY N7:92 EQU RTC:0.HR N7:93 GEQ RTC:0.MIN N7:94 BND OTE B3:3/11 EOR
%   B3:5/10  "bypass date and time reached." %
%   B3:11/9  SECONDS  "Seconds exceeded" %
%   N7:90  RTC %
%   B3:3/11  TB  "Maintence Due" %
% Rung: 31 %
SOR END EOR

OTHER DOCUMENTED ADDRESSES
  B3:10/8  "ins 8 passable"
  B38:0  EX1_GOOD
  B189:0/0  "change box"
  B189:0/9  "override boxing ok or not full signal"
  B189:0/11  "HMI force door close"
  B196:1/0  "Chute door is closed"
  B196:1/1  "control chute door"
  B196:1/13  "force box conveyor on"
  B196:3/0  "for hmi to continue production unlatched by hmi"
  HSC:0.0  "top"
  HSC:0.3/6  "Underflow interrupt"
  HSC:0.3/7  "Overflow interrupt"
  HSC:1.0  "bot"
  HSC:1.3/6  "Underflow interrupt"
  HSC:1.3/7  "Overflow interrupt"
  I7_TRAC  
  I:0.0/0  "Encoder Signal "A""
  I:0.0/4  "Encoder Signal "A""
  I:0.1/1  "spare input"
  I:0.4  "Spare Analog Input 1"
  I:0.5  "Spare Analog Input 2"
  I:0.6  "Spare Analog Input 3"
  L13:183  TKS_PER_SECOND
  L23:19  TOP_OPT_FAIL_CT
  L23:34  AIR_PRESSURE_FAULT
  L28:0  INS_1_TIME
  L29:0  INS_1_POS
  L30:0  INS_5_TIME
  L31:0  INS_5_POS
  L32:0  INS_6_TIME
  L33:0  INS_6_POS
  L192:1  BOT_LAST_TIME  "rtc bot belt previous movement event time"
  L192:2  BOT_CYCLE_TIME  "rtc bot belt time between events"
  L192:7  FROM_REAL  "distance from real part signal at optic location"
  L192:8  FROM_TRACKED  "distance from tracked part signal at optic location"
  L192:16  TOP_LAST_TIME  "rtc top belt previous movement event time"
  L192:17  TOP_CYCLE_TIME  "rtc top belt time between events"
  L199:5  ACQTM51
  L199:6  ACQTM52
  L199:7  ACQTM53
  L199:9  "ones"
  L199:10  "billions"
  L199:13  DUMP_LONG
  L199:15  ACQTM11
  L199:16  ACQTM12
  L199:17  ACQTM13
  L199:20  RESULTTM1
  L199:22  CLEARTIME5COUNT
  L199:23  CLEARTIME6COUNT
  L199:24  ACQTM61
  L199:25  ACQTM62
  L199:26  ACQTM63
  L199:27  TMSINCETRIG1
  L199:29  TMSINCETRIG5
  L199:30  TMSINCETRIG6
  L199:31  CLEARTIME1COUNT
  L199:32  RESULTTM5
  L199:33  RESULTTM6
  L199:34  MAXACQTM1
  L199:36  MAXACQTM6
  N7  
  N101:2  I3_TRIG_LOC
  N101:3  I4_TRIG_LOC
  O:0.0/1  "spare"
  PFILE:6  "check for part jams"
  PFILE:10  "Bottom belt HSC"
  PFILE:12  "Top belt HSC"
  Q2:55  END_OF_MAIN
  Q5:94  END_OF_BELTS
  T20:0  "Trigger On Time"
  U:9  "slow data"
  U:24  "check skipped fail rate"
  U:28  "faults"
  U:29  "speed"
  U:30  "count"
  U:31  "rate calc"
  U:32  "boxer"
  U:33  "bulk pack"
  U:34  "customer boxing unit signals"
  U:35  "cleanup"

COMMENTS NOT ATTACHED TO A CURRENT RUNG
  R6:2: B41 is the top good 3 file
  R6:6/DN: B35 is the top NG file
  R6:10/DN: B37 is the top good 1 file
  R6:11/DN: B39 is the top good 2 file
  B100:1/15: what is this code for?
  R6:0: B36 is the bottom GOOD file
  R6:10: B37 is the top good 1 file
  R6:6: B35 is the top NG file
  R6:4: B34 is the bottom NG file

REVISION NOTES
  13: updated count reset
  14: added io moduals
  15: multiple steps toward new hmi integration
  21: test
  27: fix error if bulk pack and no boxing fallout were on

DATA TABLE (non-zero values as saved)
DATA B3
% B3:0 % 0X88E2 0X0141 0X4000 0X5101 0X28B7 0X1504 0X1430 0X0461 0X3FC0 0X2330
% B3:10 % 0X21C0 0X40C6 0X4000 0X18D4 0X0001 0X2000 0X0000 0X0000 0X0000 0X0000
% B3:20 % 0X0100 0X0000 0X0000 0X0000 0X0000 0X0000 0X0000 0X0000 0X0000 0X0000
% B3:50 % 0X0001 0X0000 0X0000 0X0000 0X0000 0X0000 0X0000 0X0000 0X0000 0X0000
DATA T4
% .PRE .ACC %
% T4:0 % 0 3
% T4:1 % 150 0
% T4:2 % 400 0
% T4:3 % 333 215
% T4:4 % 1000 0
% T4:5 % 5 5
% T4:6 % 10 32766
% T4:7 % 150 0
% T4:8 % 20 18
% T4:9 % 50 28
% T4:10 % 200 0
% T4:11 % 400 0
% T4:12 % 40 41
% T4:13 % 250 0
% T4:14 % 666 0
% T4:15 % 1000 1001
% T4:16 % 400 0
% T4:17 % 100 65
% T4:18 % 5 0
% T4:19 % 300 0
% T4:20 % 200 0
% T4:21 % 200 0
% T4:22 % 200 0
% T4:23 % 250 0
% T4:24 % 666 0
% T4:25 % 666 0
% T4:26 % 666 0
% T4:27 % 250 0
% T4:28 % 250 0
% T4:29 % 5000 0
% T4:30 % 333 0
% T4:31 % 125 11
% T4:32 % 333 210
% T4:33 % 333 211
% T4:34 % 1111 0
% T4:35 % 23 0
% T4:36 % 5000 0
% T4:37 % 500 0
DATA C5
% .PRE .ACC %
% C5:0 % 32766 0
DATA R6
% .LEN .POS %
% R6:0 % 1250 0
% R6:1 % 16 0
% R6:2 % 1050 0
% R6:3 % 1050 0
% R6:4 % 1250 0
% R6:5 % 1250 0
% R6:6 % 1713 0
% R6:7 % 16 0
% R6:8 % 1024 0
% R6:9 % 3 0
% R6:10 % 1713 0
% R6:11 % 1050 0
% R6:12 % 10 0
% R6:13 % 10 0
% R6:14 % 10 0
% R6:15 % 10 0
% R6:16 % 1713 0
% R6:17 % 1713 0
% R6:18 % 1050 0
% R6:19 % 10 0
DATA N7
% N7:0 % 25892 5 1034 497 3 0 0 0 500 43
% N7:10 % 1000 43 0 8 22 22 1000 2000 50 1050
% N7:20 % 0 1329 16 2000 0 48 0 0 0 250
% N7:30 % 666 30173 150 0 30362 1244 78 48 0 48
% N7:40 % 6 38 1 37 145 1567 32767 1567 6 16
% N7:50 % 15 16 16 16 17 1013 0 0 73 3
% N7:60 % 1713 1713 1050 3 73 160 4999 5 400 400
% N7:70 % 100 200 300 400 90 190 290 390 -25586 24364
% N7:80 % 100 150 1263 1269 1610 1620 34 1 0 0
% N7:90 % 2011 4 4 12 1 34 1 4 250 21700
% N7:100 % 2000 90 110 100 175 25 0 0 0 0
% N7:190 % -128 27477 27605 32767 0 0 0 0 0 0
DATA F8
% F8:0 % 6
DATA L13
% L13:0 % 1202971 3570965 0 1085550 6266782
% L13:5 % 3 562059 89436 6314867 1085373
% L13:10 % 1083858 33051 0 15 90
% L13:15 % 1402079784 -2147483648 2147483647 2147483647 82058
% L13:20 % 1390108986 372254835 1200 0 100
% L13:25 % 1250356 2772910 2678505 0 1396868869
% L13:30 % 5209974 1255469 1020000 1397286388 700
% L13:35 % 0 4932407 5707357 242780359 242780388
% L13:40 % 18635 1000000000 1000000 1397286342 1397392275
% L13:45 % 1397392305 28 0 46 1390079231
% L13:50 % 4687558 89436 -50500412 0 0
% L13:55 % 4687528 26271501 13734 83784399 1398744
% L13:60 % 1109427 3990695 0 600 -1
% L13:65 % 100 -100 -207503779 -207499544 2
% L13:70 % 1379074575 45 8 1863501 1390079231
% L13:75 % 15 30 100 10974083 4
% L13:80 % 557730 74 296 40 1373440
% L13:85 % 274296 0 0 0 4687599
% L13:90 % 4687569 3 1851851 5 1397392324
% L13:95 % 679743587 344 0 1397392352 510
% L13:100 % 100 524295 -1751989696 1312119 135
% L13:105 % 510 568360 1390061372 4300 1390061363
% L13:110 % 9 1433115 367 372148306 372181353
% L13:115 % 372181361 8 4 372181357 1249997
% L13:120 % 4707523 3072 54 0 85
% L13:125 % 0 1379074575 2200 3276501 274297
% L13:130 % 235 367 389794 44588 1429953
% L13:135 % 7745 3373716 274296 1016 0
% L13:140 % 4 -4 36 5081960 106
% L13:145 % 89437 5 26271587 5 20
% L13:150 % 1572700 67108884 109530 -109530 33051
% L13:155 % 10 -10 0 28 5637628
% L13:160 % 16 49 47 132548 285213229
% L13:165 % 372181570 372181580 372181570 372181580 1055291
% L13:170 % 143889 9233 9233 1300 200
% L13:175 % -1610612220 262148 537395242 536872983 268437542
% L13:180 % -207503779 0 0 1000000 0
% L13:185 % 0 0 -207499544 0 0
% L13:190 % 0 67108896 0 134217728 65536
% L13:195 % 2165248 138543120 10 -2147352060 1207976008
% L13:200 % 100671752 4481 536871424 805324800 168855553
% L13:205 % 0 2097152 524288 5907910 4886293
% L13:210 % -2111790848 4210696 4194320 65536 1048608
% L13:215 % 136314880 262145 35655680 1589280 0
% L13:220 % 16 0 4096 50332160 71303296
% L13:225 % 1073741824 1049600 1107296257 8192 -2113929216
% L13:230 % 33560576 256 1141374976 1024 -2147483584
% L13:235 % 0 270532608 8 262144 2
% L13:240 % 0 0 262144 65536 128
% L13:245 % 0 2097156 1024 268996608 -2071985920
% L13:250 % 16777216 2097152 262160 0 0
DATA L19
% L19:0 % 1396875757 1396882732 1396889965 1396897910 1396904539
% L19:5 % 1396911820 1396918817 1396926136 1396932903 1396941355
% L19:10 % 1396949074 1396955983 1396963010 1397371989 1397382389
% L19:15 % 1397391623 1396868869 16777216 256 262144
% L19:20 % 4 0 0 0 0
% L19:25 % 0 1376256 4096 8 33652736
% L19:30 % 131072 524288 -2147483648 0 -2147483648
% L19:35 % 0 0 84 0 32768
% L19:40 % 0 4096 1073741824 0 0
% L19:45 % 256 0 0 16 5250
DATA L20
% L20:0 % 1334350049 1334365823 1334403407 1336798316 1396589883
% L20:5 % 1396599679 1396777581 1396790496 1396838510 1396845576
% L20:10 % 1396853674 1396862598 1396869521 1396876409 1396883385
% L20:15 % 1396890616 1396898561 1396905190 1396912471 1396919470
% L20:20 % 1396926788 1396933557 1396942006 1396949725 1396956635
% L20:25 % 1396963662 1397284445 1397284787 1397285131 1397285469
% L20:30 % 1397285809 1397286151 1397286492 1397383042 1397392275
% L20:35 % 1328845477 1328845816 1328846153 1328846491 1328846830
% L20:40 % 1328847168 1328847507 1328847845 1328848183 1328848521
% L20:45 % 1328848858 1328849196 1328849534 1328849873 1328850210
% L20:50 % 1328850548 1328850886 1328851225 1328851563 1328851900
% L20:55 % 1328852238 1328852576 1328852915 1328853253 1328853591
% L20:60 % 1328853927 1328854266 1328854604 1328854942 1328855282
% L20:65 % 1328855619 1328855956 1328856293 1328856631 1328856968
% L20:70 % 1328857306 1328857643 1328857981 1328858319 1328858658
% L20:75 % 1328858996 1328859334 1328859672 1328860009 1328860348
% L20:80 % 1328860685 1328861024 1328861361 1328861699 1328862037
% L20:85 % 1328862375 1328862714 1328863053 1328863391 1328863729
% L20:90 % 1328864066 1328864404 1328864743 1328865081 1328865419
% L20:95 % 1328865758 1328866095 1328879445 1334259221 1334330859
% L20:100 % 33554432 37224448 1073751040 536870914 0
% L20:105 % 0 1 1057 0 0
% L20:110 % 33554432 1024 0 0 0
% L20:115 % 0 0 134219777 112 1073741824
% L20:120 % 16777216 2097152 32896 1073752096 134479876
% L20:125 % 16512 32768 68157444 84934656 0
% L20:130 % 1073741824 12582912 67112960 536873088 67109120
% L20:135 % 772 67109008 4096 67108864 8408096
% L20:140 % 67108864 536891393 268435456 4194592 1048832
% L20:145 % 8390672 33024 2129920 33557056 268435456
% L20:150 % 268435456 262656 16777216 0 10
% L20:155 % 32768 1 0 1048960 0
% L20:160 % 134217728 0 0 134217728 16777472
% L20:165 % 524352 0 1 0 131072
% L20:170 % 536870912 2195457 0 262144 0
% L20:175 % 65536 0 268435456 16384 1048576
% L20:180 % 0 16 0 0 1073743872
% L20:185 % 4456448 0 67108880 75497472 16384
% L20:190 % 512 -2013265920 131106 -2147463168 -2112880640
% L20:195 % 4098 84017472 2101780 8 272761088
% L20:200 % 514 67109376 67141632 0 2048
% L20:205 % 536870912 67108864 32768 0 2
% L20:210 % 8650752 0 16 8388608 0
% L20:215 % -2147482624 134217728 8 16384 0
% L20:220 % 67108866 1074268160 0 32 -2139095040
% L20:225 % 16777216 256 67108864 4194320 2048
% L20:230 % 272630016 0 1073774592 -2147483644 4
% L20:235 % 3146304 8262 65600 16777344 262144
% L20:240 % 1024 134217728 68 4160 1073750528
% L20:245 % 1073741824 268500992 0 285212676 824184832
% L20:250 % 4096 262400 134219776 8192 4096
% L20:255 % 1073774592
DATA L21
% L21:0 % 370126376 370131623 370144124 370940781 371914637
% L21:5 % 371917896 371977085 371981382 371997356 371999706
% L21:10 % 372002400 372005369 372007672 372009963 372012283
% L21:15 % 372014689 372017332 372019537 372021960 372024288
% L21:20 % 372026722 372028974 372031784 372034352 372036651
% L21:25 % 372038989 372145697 372145811 372145925 372146038
% L21:30 % 372146151 372146264 372146378 372178498 372181570
% L21:35 % 368302812 368302812 368302812 368302812 368302812
% L21:40 % 368302812 368302812 368302812 368302812 368302812
% L21:45 % 368302812 368302812 368302812 368302812 368302812
% L21:50 % 368302812 368302812 368302812 368302812 368302812
% L21:55 % 368302812 368302812 368302812 368302812 368302812
% L21:60 % 368302812 368302812 368302812 368302812 368302812
% L21:65 % 368302812 368302812 368302812 368302812 368302812
% L21:70 % 368302812 368302812 368302812 368302812 368302812
% L21:75 % 368302812 368302812 368302812 368302812 368302812
% L21:80 % 368302812 368302812 368302812 368302812 368302812
% L21:85 % 368302812 368302812 368302812 368302812 368302812
% L21:90 % 368302812 368302812 368302812 368302812 368302812
% L21:95 % 368302812 368302812 368306584 370096159 370119992
% L21:100 % 32 83886080 1094746112 20480 -2143289344
% L21:105 % 1073741856 65536 0 4174 543162960
% L21:110 % 263274 4224 67108872 134479872 -2147479472
% L21:115 % 536870912 39168 364544 149512 18564
% L21:120 % 1127432 537395200 268352 67109384 1024
% L21:125 % 4096 -2147483648 1 131072 1
% L21:130 % 8 1048576 0 -2139094080 18875272
% L21:135 % 416 7425 603981440 67110528 138016
% L21:140 % 33556096 1073749014 5776064 50355200 39488
% L21:145 % 8814849 8478720 -2147106560 -2012807168 3671296
% L21:150 % 5390464 2752512 20971553 532480 1078722560
% L21:155 % 128 33554433 1024 4196360 1344012289
% L21:160 % 1207959872 8429584 33554435 1080033282 656128
% L21:165 % 268435456 524352 -2139094008 704692248 134218020
% L21:170 % 134225924 0 704512 -2147445760 43008
% L21:175 % 134294528 32 1073741832 2097286 1049088
% L21:180 % 16908968 101711874 131072 10756096 1073774740
% L21:185 % 33554688 786560 0 135204 50364416
% L21:190 % 33554496 -1609562624 268456960 262144 8192
% L21:195 % 1073741824 268435456 131072 0 524808
% L21:200 % 2097152 2097152 2432 0 1048576
% L21:205 % 16777728 526688 67108880 5378080 8704
% L21:210 % 33554432 2097153 4366336 704718849 36131460
% L21:215 % 1572864 1266698272 12583040 -1555038208 18690
% L21:220 % 512 134217876 1073872896 5120 1073741824
% L21:225 % 0 335609920 16 -2147483646 524288
% L21:230 % 68157472 80 4194304 134221824 67109248
% L21:235 % 134217728 134217728 537952256 603979776 16387
% L21:240 % 2949269 688128 1494239520 4194304 38535172
% L21:245 % 1073742226 33587348 67125289 2048 536870912
% L21:250 % -2147466238 65536 1879261186 67108931 5507744
% L21:255 % 1
DATA L22
% L22:0 % 1397383072 1397392305 1328699186 1328699525 1328699864
% L22:5 % 1328700203 1328700541 1328700881 1328701220 1328701560
% L22:10 % 1328701900 1328702242 1328702585 1328716716 1328879475
% L22:15 % 1334259251 1334330889 1334350079 1334365853 1334403437
% L22:20 % 1336798346 1396589914 1396599709 1396777611 1396790526
% L22:25 % 1396838540 1396845607 1396853704 1396862629 1396869551
% L22:30 % 1396876438 1396883415 1396890646 1396898591 1396905220
% L22:35 % 1396912501 1396919500 1396926818 1396933586 1396942036
% L22:40 % 1396949755 1396956665 1396963692 1397284520 1397284859
% L22:45 % 1397285200 1397285542 1397285881 1397286221 1397286560
DATA L23
% L23:0 % 372178508 372181580 368281741 368281741 368281741
% L23:5 % 368281741 368281741 368281761 368281816 368281893
% L23:10 % 368281983 368282082 368282185 368286906 368306594
% L23:15 % 370096169 370120002 370126386 370131633 370144134
% L23:20 % 370940791 371914647 371917906 371977095 371981392
% L23:25 % 371997366 371999716 372002410 372005379 372007682
% L23:30 % 372009973 372012293 372014699 372017342 372019547
% L23:35 % 372021970 372024298 372026732 372028984 372031794
% L23:40 % 372034362 372036661 372038999 372145722 372145834
% L23:45 % 372145948 372146062 372146175 372146288 372146400
DATA L30
% L30:0 % 1322623720 1322635911 1322651160 1322657604 1322669674
% L30:5 % 1322681773 1322695117 1322707231 1322720149 1322732730
% L30:10 % 1322746238 1322760397 1322773078 1322784830 1322797133
% L30:15 % 1322809833 1326622778 1326638116 1326652841 1326672550
% L30:20 % 1326687651 1326784122 1327328979 1327329318 1327329656
% L30:25 % 1327329995 1327330334 1327330671 1327331011 1328045707
% L30:30 % 1328058182 1328395590 1328710104 1328872957 1334252638
% L30:35 % 1334324287 1334343468 1334359234 1334395660 1334395999
% L30:40 % 1396770994 1396783915 1397284293 1397284633 1397284974
% L30:45 % 1397285316 1397285657 1397285998 1397286342 1322605738
DATA L31
% L31:0 % 1386621470 1386625527 1386630600 1386632742 1386636759
% L31:5 % 1386640785 1386645224 1386649253 1386653550 1386657736
% L31:10 % 1386662229 1386666939 1386671159 1386675068 1386679162
% L31:15 % 1386683385 1387951791 1387956893 1387961790 1387968345
% L31:20 % 1387973369 1388005463 1388015611 1388015611 1388015611
% L31:25 % 1388015611 1388015611 1388015611 1388015611 1388018565
% L31:30 % 1388022716 1388134956 1388153045 1388172699 1389962245
% L31:35 % 1389986078 1389992459 1389997704 1390009819 1390009932
% L31:40 % 1390057198 1390061497 1390078549 1390078662 1390078775
% L31:45 % 1390078889 1390079002 1390079116 1390079231 1386615491
DATA L32
% L32:0 % 10973377 10973506 10973641 10973772 10973903
% L32:5 % 10974038 -50500412 -50500276 -50500145 -50500013
% L32:10 % -50499883 -50499747 -50499616 -50499484 -50499350
% L32:15 % -50499219 -50499082 -50498952 -50498822 -50498691
% L32:20 % -50498561 -50498425 10969253 10969386 10969516
% L32:25 % 10969648 10969779 10969912 10970043 10970176
% L32:30 % 10970307 10970438 10970571 10970705 10970835
% L32:35 % 10970966 10971096 10971228 10971363 10971929
% L32:40 % 10972065 10972197 10972327 10972458 10972587
% L32:45 % 10972718 10972850 10972986 10973116 10973247
DATA L33
% L33:0 % 1379074448 1379074473 1379074499 1379074524 1379074549
% L33:5 % 1379074575 1367302347 1367302373 1367302398 1367302423
% L33:10 % 1367302448 1367302474 1367302499 1367302524 1367302550
% L33:15 % 1367302575 1367302601 1367302626 1367302651 1367302676
% L33:20 % 1367302701 1367302727 1379073659 1379073684 1379073709
% L33:25 % 1379073734 1379073759 1379073785 1379073810 1379073835
% L33:30 % 1379073861 1379073886 1379073911 1379073937 1379073962
% L33:35 % 1379073987 1379074011 1379074037 1379074063 1379074171
% L33:40 % 1379074197 1379074222 1379074247 1379074272 1379074297
% L33:45 % 1379074322 1379074347 1379074373 1379074398 1379074423
DATA B34
% B34:80 % 0X0200 0X0800 0X0000 0X4000 0X0040 0X5000 0X0000 0X0000 0X0100 0X8000
% B34:90 % 0X0080 0X0000 0X8400 0X0000 0X0000 0X8000 0X0000 0X0000 0X4000 0X0000
% B34:100 % 0X0000 0X0000 0X8000 0X0000 0X0000 0X0002 0X0000 0X0000 0X0000 0X0200
% B34:110 % 0X0000 0X0400 0X0000 0X0000 0X0000 0X0000 0X0220 0X0000 0X0100 0X0000
% B34:120 % 0X0000 0X0000 0X0000 0X1000 0X0000 0X0000 0X0000 0X8020
DATA B35
% B35:110 % 0X0000 0X0000 0X0200 0X0000 0X0000 0X0000 0X0000 0X0000 0X0000 0X0000
DATA B37
% B37:0 % 0X0000 0X0000 0X2000 0X0000 0X0000 0X0000 0X0000 0X0000 0X0000 0X0000
DATA B40
% B40:0 % 0XAAAA
DATA B41
% B41:60 % 0X0000 0X0000 0X0000 0X0000 0X1E00 0X0000 0X0000 0X0000 0X0000 0X0000
DATA B100
% B100:0 % 0X0700 0X1800 0X8024 0X0000 0X0000 0X0000 0X0000 0X0000 0X0000 0X0000
DATA N101
% N101:0 % 130 646 0 0 1178 100 1030 1200 1200 1243
% N101:10 % 1253 1530 10 15727 778 17365 1589 333 333 125
% N101:20 % 1000 500 400 0 0 0 333 333 0 0
DATA L102
% L102:0 % 40 8 1 1 3300
% L102:5 % 3300 0 0 0 0
% L102:10 % 0 1 0 0 1851851
% L102:15 % 0 30 18 30 19
% L102:20 % 0 13 0 0 49
% L102:25 % 46 0 1 495 0
% L102:30 % 45 0 25429776 0 -12977701
% L102:35 % 0 50000 0 999999 47
% L102:40 % 0 2 0 0 17
DATA A190
% A190:0 % 0X3C21 0X4142 0X4344 0X4D2D 0X3230 0X3E0D 0X0A3C 0X6874 0X6D6C 0X3E0D
% A190:10 % 0X0A3C 0X626F 0X6479 0X3E0D 0X0A0D 0X0A3C 0X2141 0X4244 0X5452 0X2D4E
% A190:20 % 0X3130 0X313A 0X312C 0X3130 0X214C 0X6973 0X7420 0X6F66 0X2043 0X7572
% A190:30 % 0X7265 0X6E74 0X2054 0X656D 0X7065 0X7261 0X7475 0X7265 0X2072 0X6561
% A190:40 % 0X6469 0X6E67 0X733E 0X0D0A 0X0D0A 0X0D0A 0X3C21 0X4142 0X4454 0X522D
% A190:50 % 0X4E37 0X3A30 0X2C31 0X2154 0X6573 0X7469 0X6E67 0X3E0D 0X0A0D 0X0A54
% A190:60 % 0X6869 0X7320 0X7465 0X7874 0X2068 0X6572 0X6520 0X646F 0X6573 0X6E27
% A190:70 % 0X7420 0X7368 0X6F77 0X2075 0X703F 0X200D 0X0A0D 0X0A3C 0X2F62 0X6F64
% A190:80 % 0X793E 0X0D0A 0X3C2F 0X6874 0X6D6C 0X3E00 0X7464 0X3E0D 0X0A3C 0X7464
% A190:90 % 0X3E3C 0X2141 0X4244 0X5452 0X2D6E 0X7B31 0X3031 0X7D3A 0X7B31 0X367D
% A190:100 % 0X3E3C 0X2F74 0X643E 0X0D0A 0X3C2F 0X7472 0X3E0D 0X0A3C 0X2F74 0X6162
% A190:110 % 0X6C65 0X3E0D 0X0A3C 0X2F62 0X6F64 0X793E 0X0D0A 0X3C2F 0X6874 0X6D6C
% A190:120 % 0X3E00 0X0000 0X0000 0X0000 0X0000 0X0000 0X0000 0X0000 0X0000 0X0000
